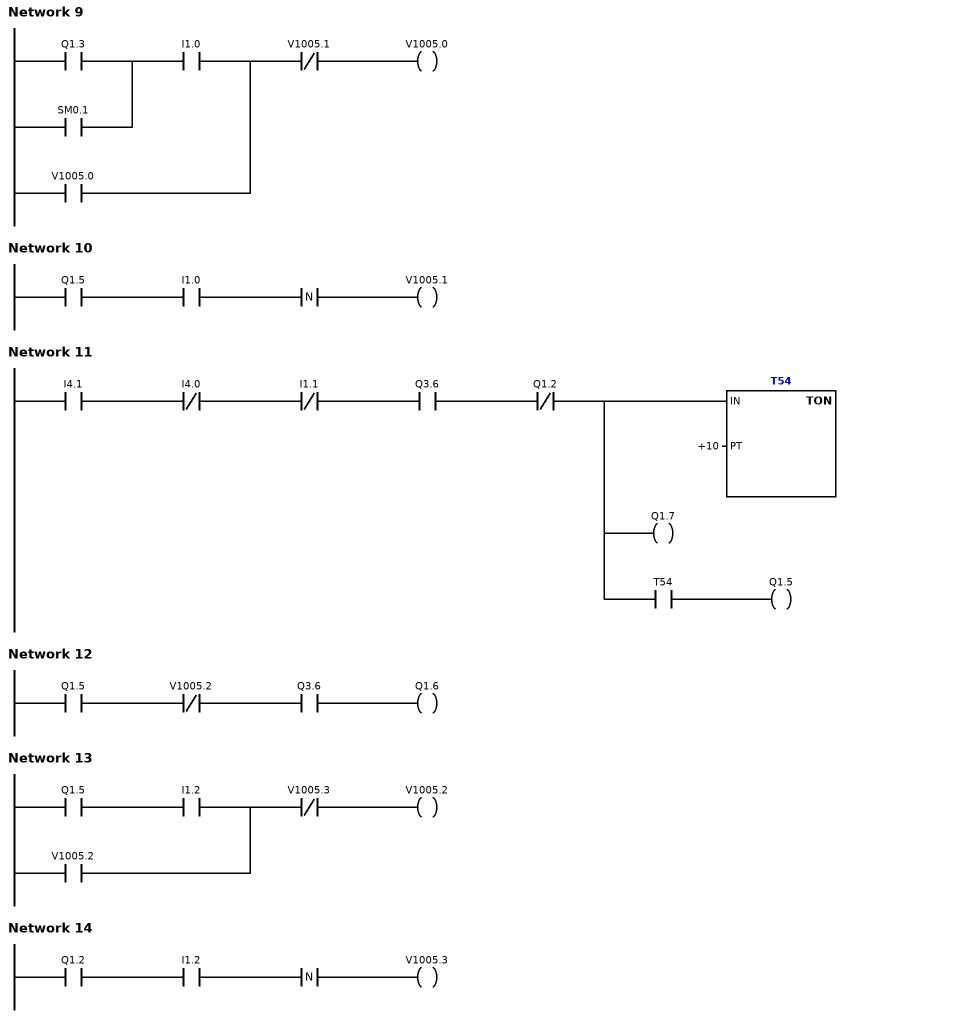
[picture p24: SBR7 networks 9-14]
Network 9
LD     Q1.3
O      SM0.1
A      I1.0
O      V1005.0
AN     V1005.1
=      V1005.0
Network 10
LD     Q1.5
A      I1.0
ED
=      V1005.1
Network 11
LD     I4.1
AN     I4.0
AN     I1.1
A      Q3.6
AN     Q1.2
TON    T54, +10
=      Q1.7
A      T54
=      Q1.5
Network 12
LD     Q1.5
AN     V1005.2
A      Q3.6
=      Q1.6
Network 13
LD     Q1.5
A      I1.2
O      V1005.2
AN     V1005.3
=      V1005.2
Network 14
LD     Q1.2
A      I1.2
ED
=      V1005.3
END_SUBROUTINE_BLOCK

SUBROUTINE_BLOCK Sheed_lead:SBR8
TITLE=
BEGIN
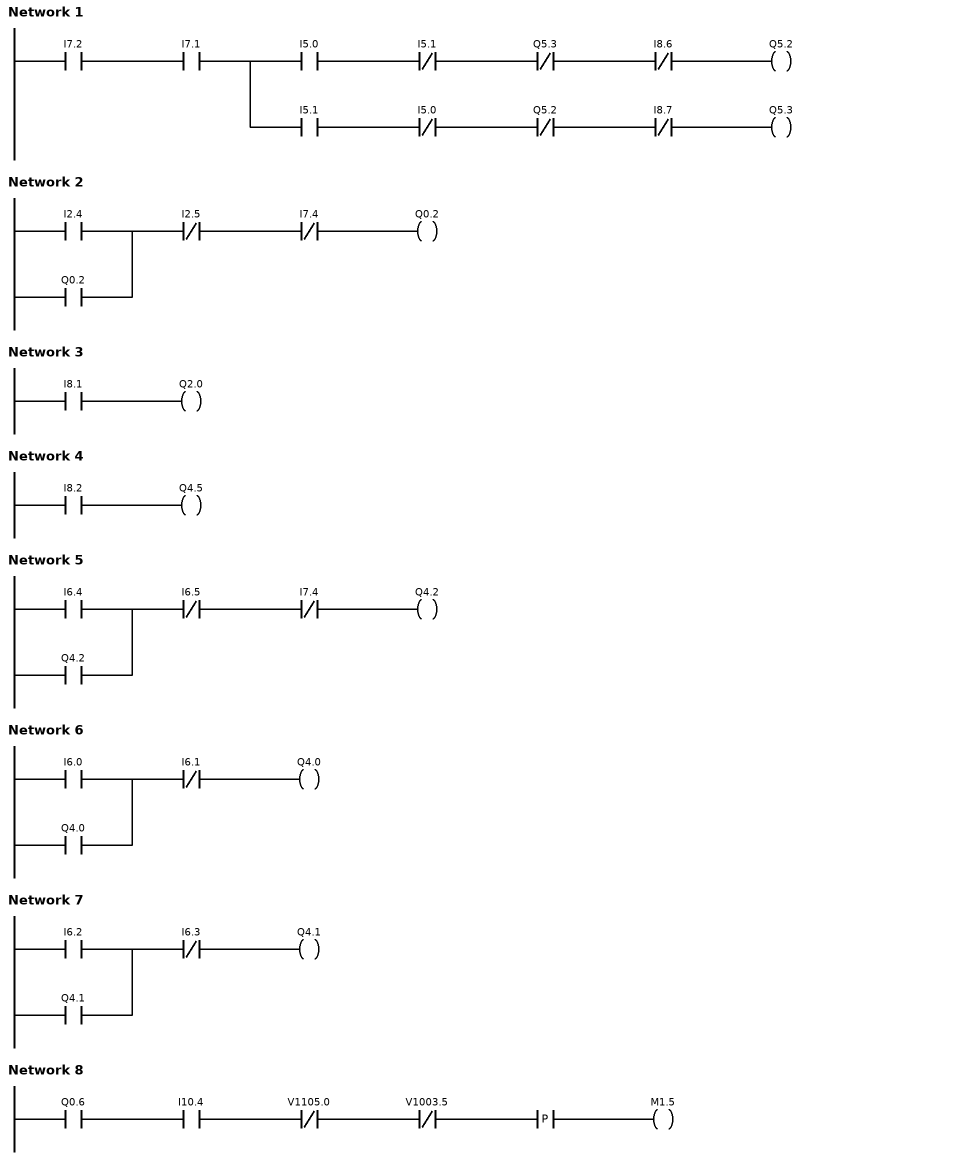
Network 1
LD     I7.2
A      I7.1
LPS
A      I5.0
AN     I5.1
AN     Q5.3
AN     I8.6
=      Q5.2
LPP
A      I5.1
AN     I5.0
AN     Q5.2
AN     I8.7
=      Q5.3
Network 2
LD     I2.4
O      Q0.2
AN     I2.5
AN     I7.4
=      Q0.2
Network 3
LD     I8.1
=      Q2.0
Network 4
LD     I8.2
=      Q4.5
Network 5
LD     I6.4
O      Q4.2
AN     I6.5
AN     I7.4
=      Q4.2
Network 6
LD     I6.0
O      Q4.0
AN     I6.1
=      Q4.0
Network 7
LD     I6.2
O      Q4.1
AN     I6.3
=      Q4.1
Network 8
LD     Q0.6
A      I10.4
AN     V1105.0
AN     V1003.5
EU
=      M1.5
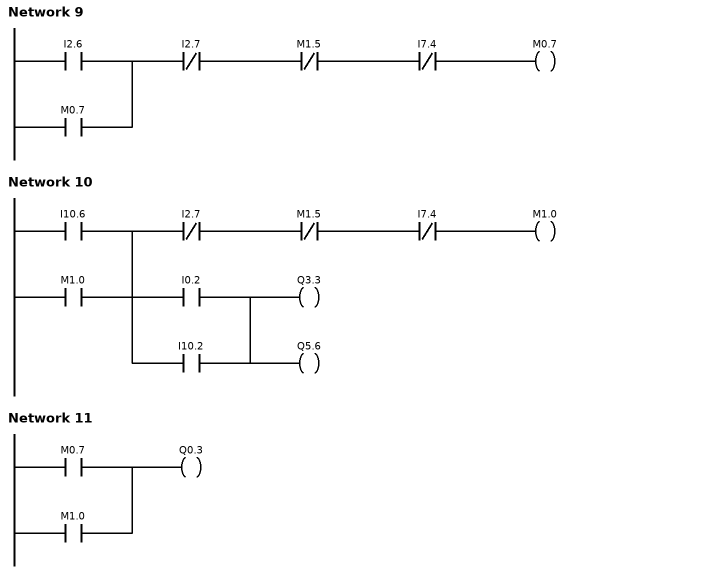
Network 9
LD     I2.6
O      M0.7
AN     I2.7
AN     M1.5
AN     I7.4
=      M0.7
Network 10
LD     I10.6
O      M1.0
LPS
AN     I2.7
AN     M1.5
AN     I7.4
=      M1.0
LPP
LD     I0.2
O      I10.2
ALD
=      Q3.3
=      Q5.6
Network 11
LD     M0.7
O      M1.0
=      Q0.3
END_SUBROUTINE_BLOCK

SUBROUTINE_BLOCK Core_Chuck:SBR9
TITLE=
BEGIN
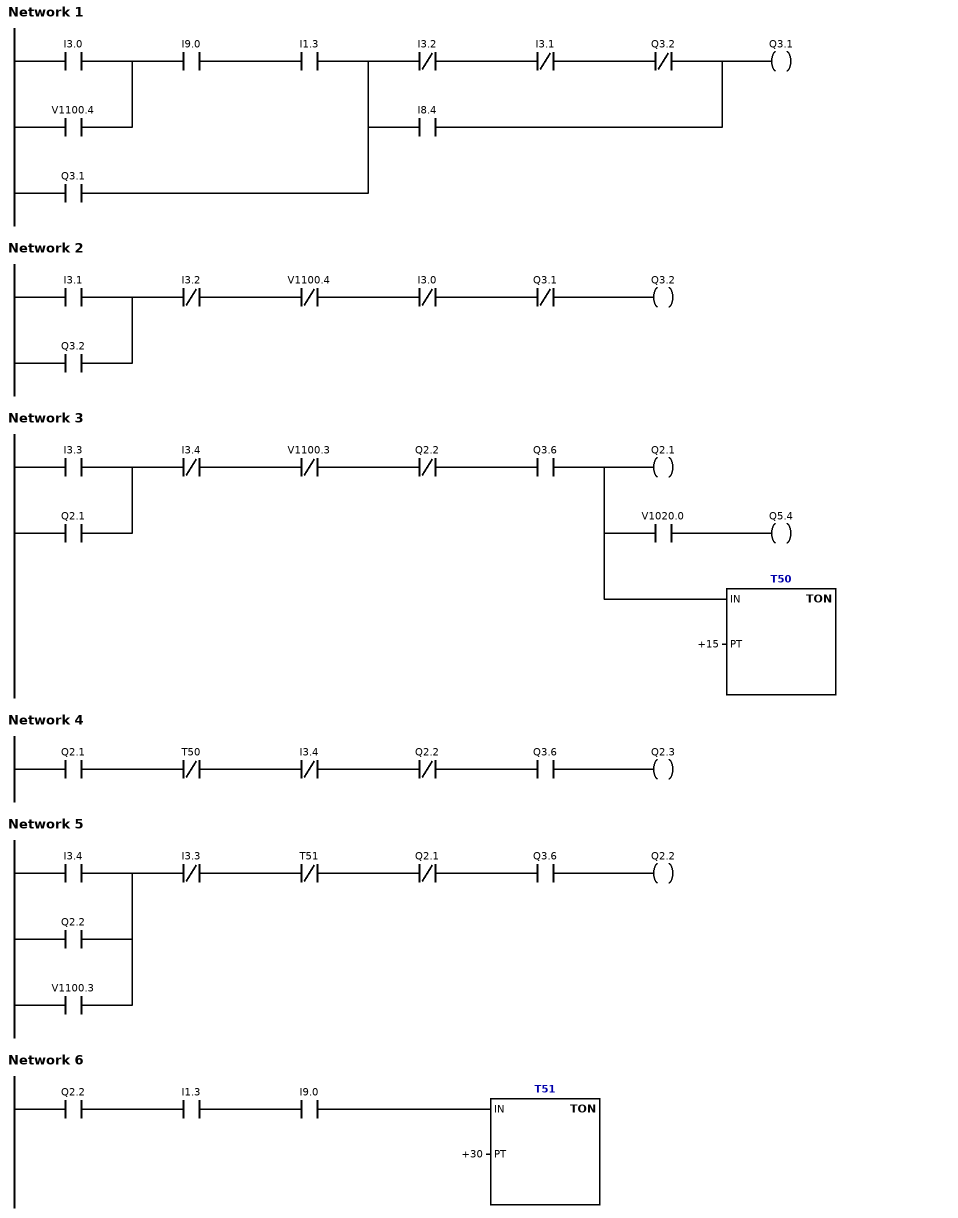
Network 1
LD     I3.0
O      V1100.4
A      I9.0
A      I1.3
O      Q3.1
LDN    I3.2
AN     I3.1
AN     Q3.2
O      I8.4
ALD
=      Q3.1
Network 2
LD     I3.1
O      Q3.2
AN     I3.2
AN     V1100.4
AN     I3.0
AN     Q3.1
=      Q3.2
Network 3
LD     I3.3
O      Q2.1
AN     I3.4
AN     V1100.3
AN     Q2.2
A      Q3.6
LPS
=      Q2.1
A      V1020.0
=      Q5.4
LPP
TON    T50, +15
Network 4
LD     Q2.1
AN     T50
AN     I3.4
AN     Q2.2
A      Q3.6
=      Q2.3
Network 5
LD     I3.4
O      Q2.2
O      V1100.3
AN     I3.3
AN     T51
AN     Q2.1
A      Q3.6
=      Q2.2
Network 6
LD     Q2.2
A      I1.3
A      I9.0
TON    T51, +30
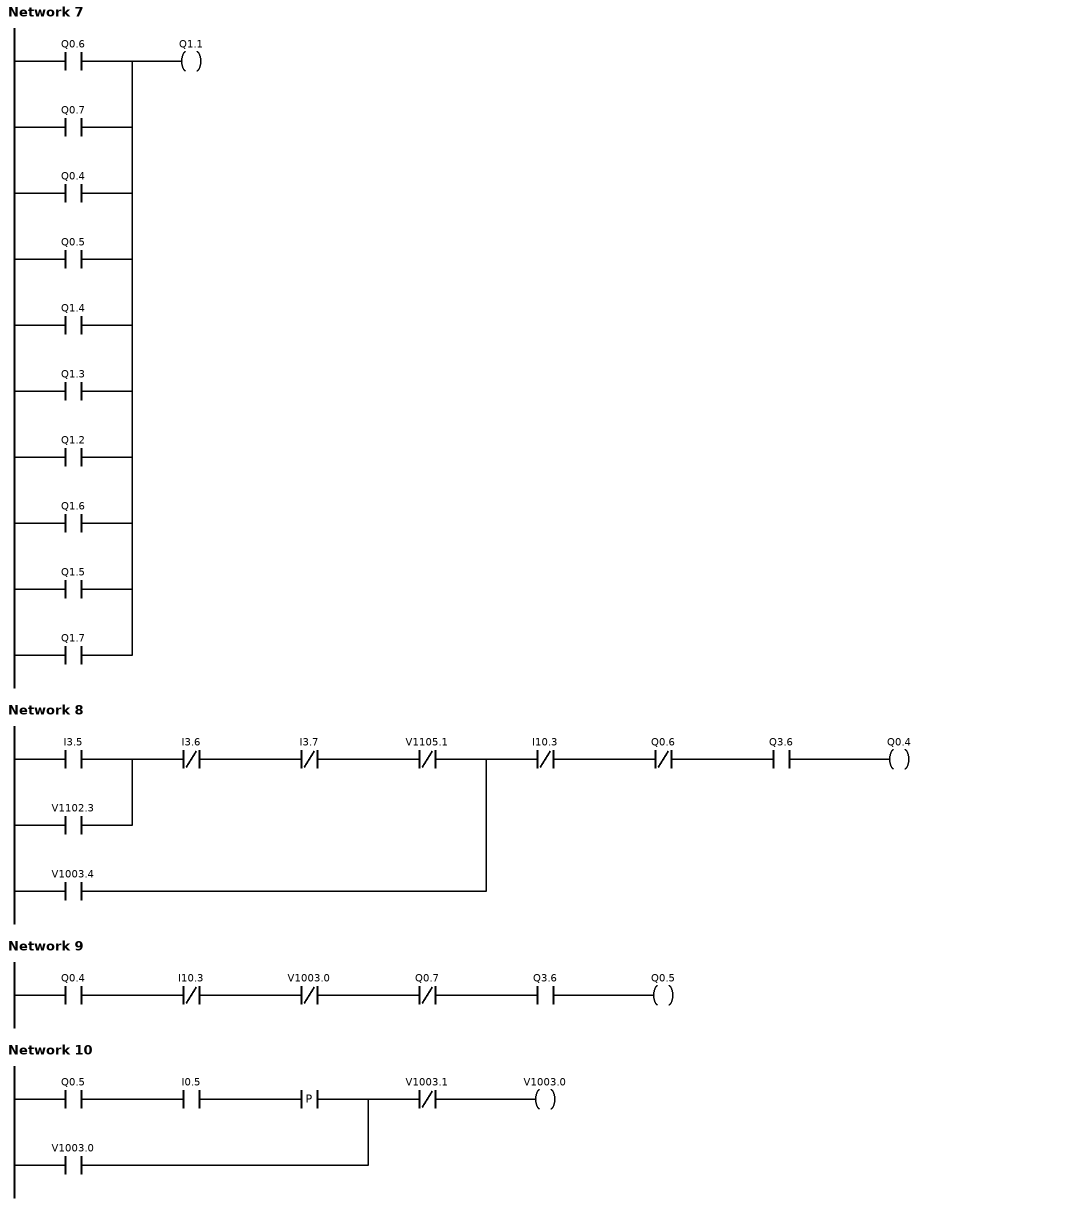
Network 7
LD     Q0.6
O      Q0.7
O      Q0.4
O      Q0.5
O      Q1.4
O      Q1.3
O      Q1.2
O      Q1.6
O      Q1.5
O      Q1.7
=      Q1.1
Network 8
LD     I3.5
O      V1102.3
AN     I3.6
AN     I3.7
AN     V1105.1
O      V1003.4
AN     I10.3
AN     Q0.6
A      Q3.6
=      Q0.4
Network 9
LD     Q0.4
AN     I10.3
AN     V1003.0
AN     Q0.7
A      Q3.6
=      Q0.5
Network 10
LD     Q0.5
A      I0.5
EU
O      V1003.0
AN     V1003.1
=      V1003.0
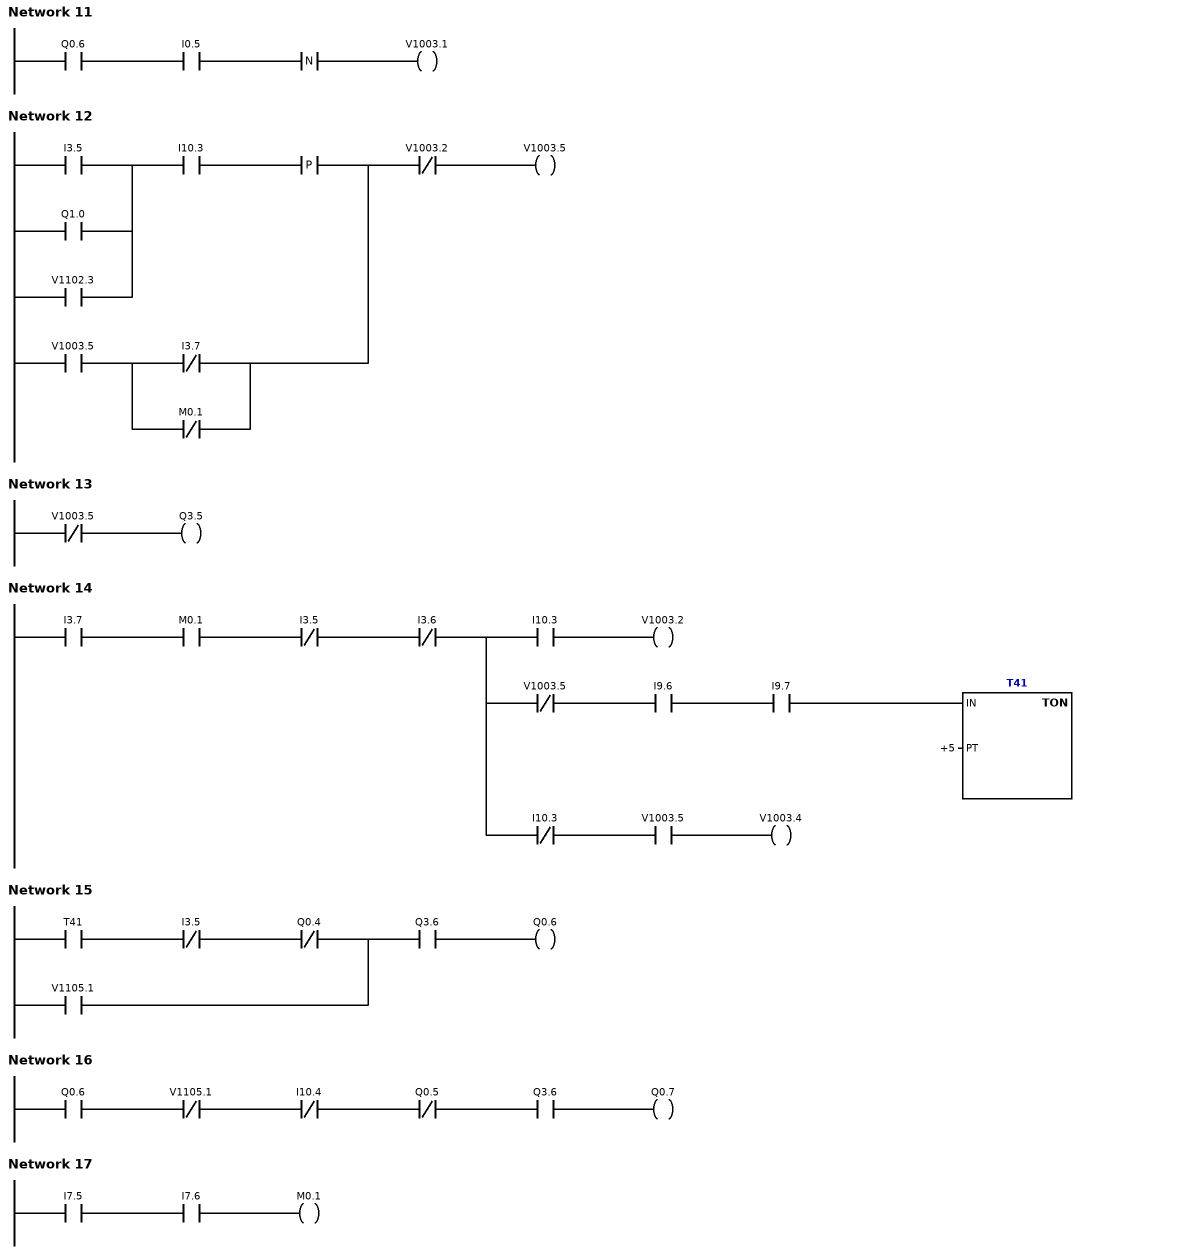
Network 11
LD     Q0.6
A      I0.5
ED
=      V1003.1
Network 12
LD     I3.5
O      Q1.0
O      V1102.3
A      I10.3
EU
LD     V1003.5
LDN    I3.7
ON     M0.1
ALD
OLD
AN     V1003.2
=      V1003.5
Network 13
LDN    V1003.5
=      Q3.5
Network 14
LD     I3.7
A      M0.1
AN     I3.5
AN     I3.6
LPS
A      I10.3
=      V1003.2
LRD
AN     V1003.5
A      I9.6
A      I9.7
TON    T41, +5
LPP
AN     I10.3
A      V1003.5
=      V1003.4
Network 15
LD     T41
AN     I3.5
AN     Q0.4
O      V1105.1
A      Q3.6
=      Q0.6
Network 16
LD     Q0.6
AN     V1105.1
AN     I10.4
AN     Q0.5
A      Q3.6
=      Q0.7
Network 17
LD     I7.5
A      I7.6
=      M0.1
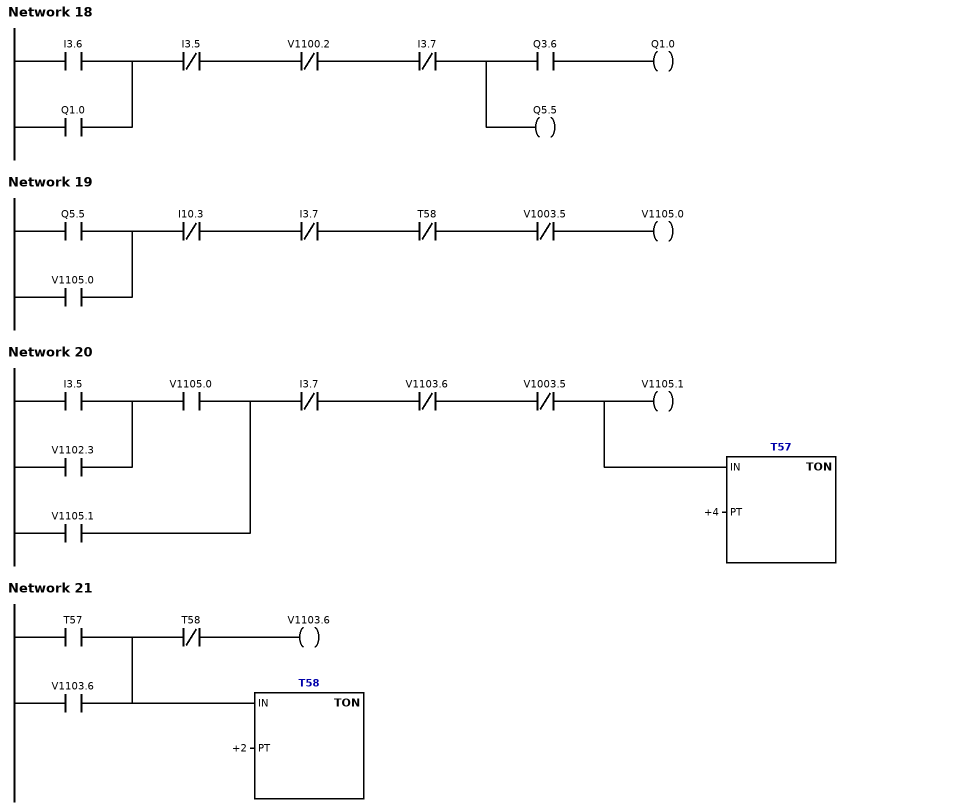
Network 18
LD     I3.6
O      Q1.0
AN     I3.5
AN     V1100.2
AN     I3.7
LPS
A      Q3.6
=      Q1.0
LPP
=      Q5.5
Network 19
LD     Q5.5
O      V1105.0
AN     I10.3
AN     I3.7
AN     T58
AN     V1003.5
=      V1105.0
Network 20
LD     I3.5
O      V1102.3
A      V1105.0
O      V1105.1
AN     I3.7
AN     V1103.6
AN     V1003.5
=      V1105.1
TON    T57, +4
Network 21
LD     T57
O      V1103.6
LPS
AN     T58
=      V1103.6
LPP
TON    T58, +2
END_SUBROUTINE_BLOCK

SUBROUTINE_BLOCK Value_1:SBR10
TITLE=
VAR_INPUT
d1:REAL;	// LD0 
H:REAL;	// LD4 
END_VAR
VAR_OUTPUT
D:REAL;	// LD8 
END_VAR
BEGIN
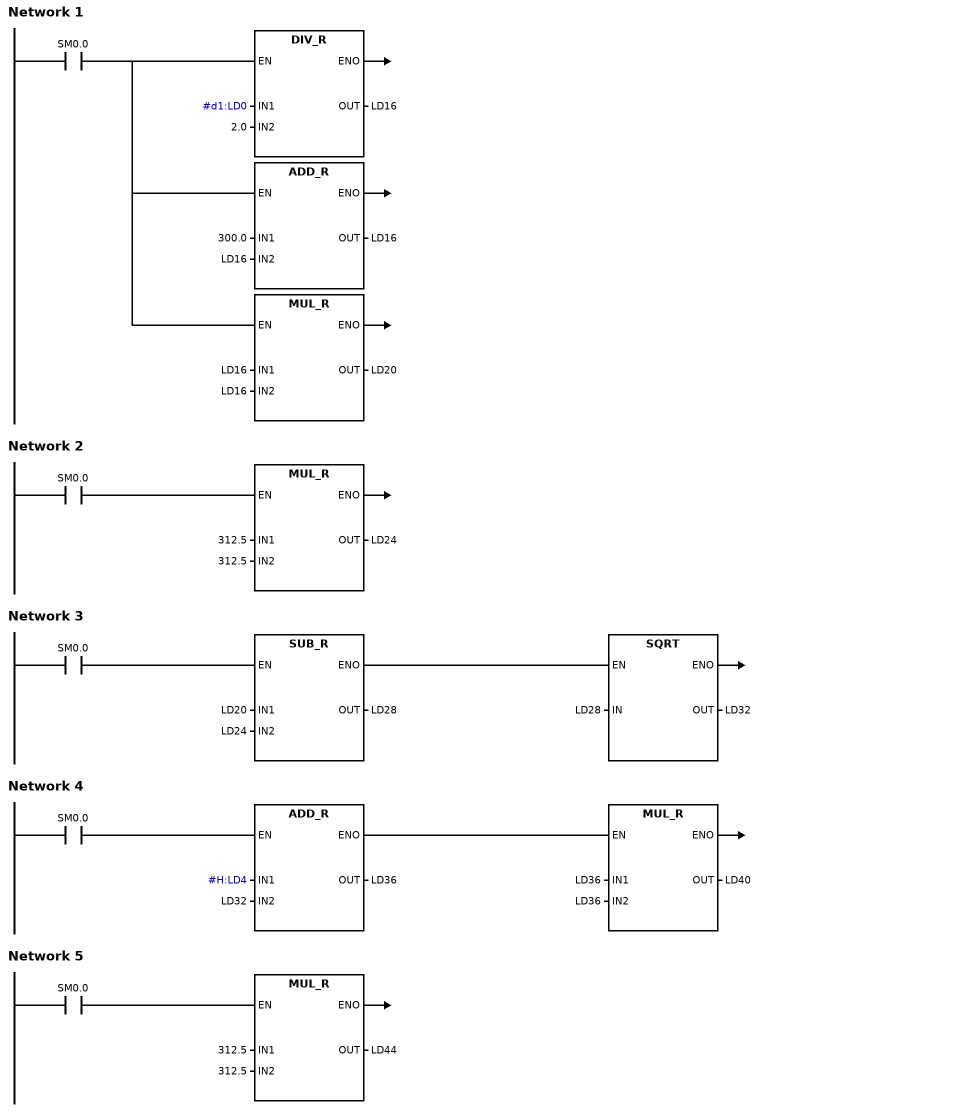
Network 1
LD     SM0.0
MOVR   #d1:LD0, LD16
/R     2.0, LD16
+R     300.0, LD16
MOVR   LD16, LD20
*R     LD16, LD20
Network 2
LD     SM0.0
MOVR   312.5, LD24
*R     312.5, LD24
Network 3
LD     SM0.0
MOVR   LD20, LD28
AENO
-R     LD24, LD28
AENO
SQRT   LD28, LD32
Network 4
LD     SM0.0
MOVR   #H:LD4, LD36
AENO
+R     LD32, LD36
AENO
MOVR   LD36, LD40
*R     LD36, LD40
Network 5
LD     SM0.0
MOVR   312.5, LD44
*R     312.5, LD44
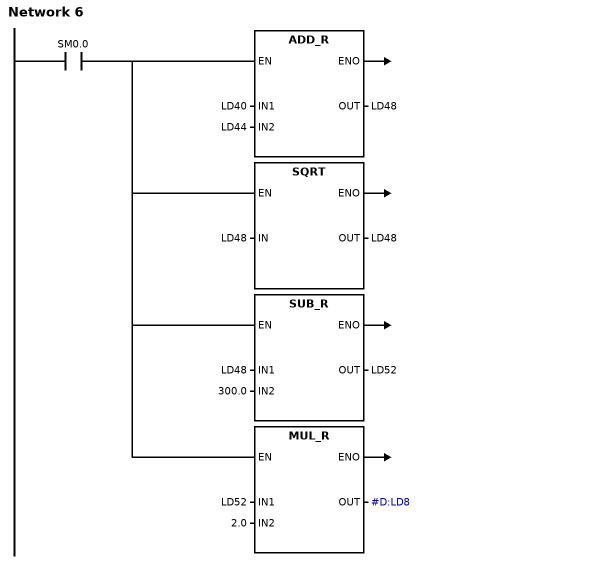
Network 6
LD     SM0.0
MOVR   LD40, LD48
+R     LD44, LD48
SQRT   LD48, LD48
MOVR   LD48, LD52
-R     300.0, LD52
MOVR   LD52, #D:LD8
*R     2.0, #D:LD8
END_SUBROUTINE_BLOCK

SUBROUTINE_BLOCK TOSHIBA_DO:SBR11
TITLE=
BEGIN
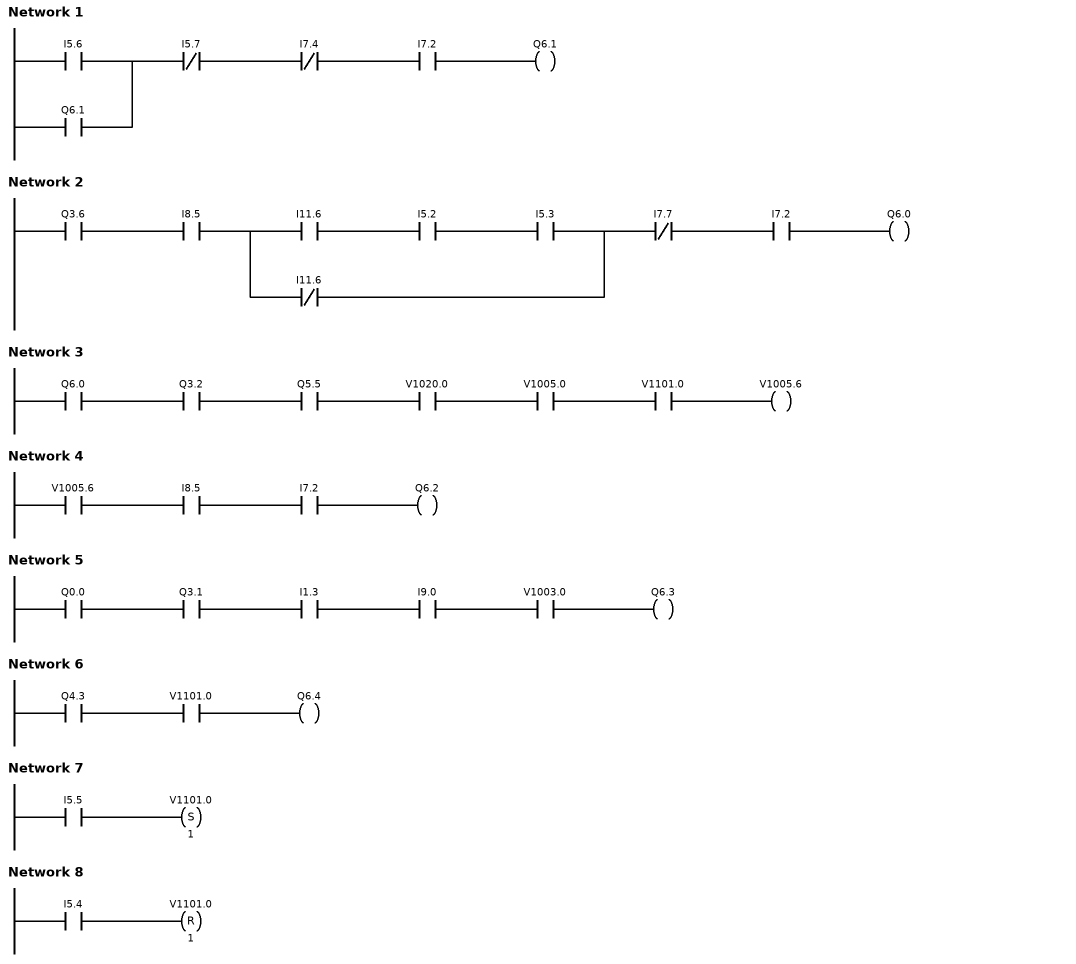
Network 1
LD     I5.6
O      Q6.1
AN     I5.7
AN     I7.4
A      I7.2
=      Q6.1
Network 2
LD     Q3.6
A      I8.5
LD     I11.6
A      I5.2
A      I5.3
ON     I11.6
ALD
AN     I7.7
A      I7.2
=      Q6.0
Network 3
LD     Q6.0
A      Q3.2
A      Q5.5
A      V1020.0
A      V1005.0
A      V1101.0
=      V1005.6
Network 4
LD     V1005.6
A      I8.5
A      I7.2
=      Q6.2
Network 5
LD     Q0.0
A      Q3.1
A      I1.3
A      I9.0
A      V1003.0
=      Q6.3
Network 6
LD     Q4.3
A      V1101.0
=      Q6.4
Network 7
LD     I5.5
S      V1101.0, 1
Network 8
LD     I5.4
R      V1101.0, 1
END_SUBROUTINE_BLOCK

SUBROUTINE_BLOCK Auto_Roll_Eiector:SBR12
TITLE=
BEGIN
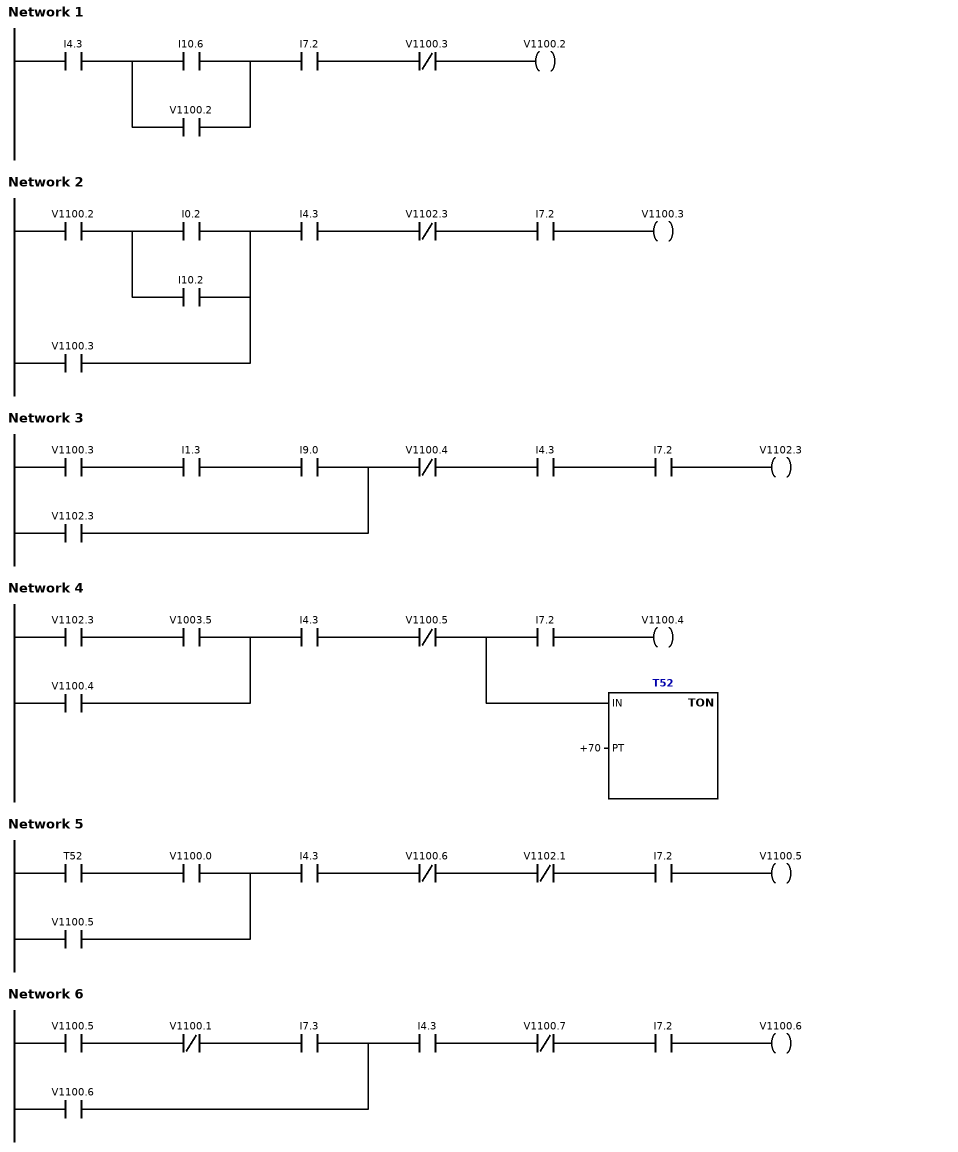
Network 1
LD     I4.3
LD     I10.6
O      V1100.2
ALD
A      I7.2
AN     V1100.3
=      V1100.2
Network 2
LD     V1100.2
LD     I0.2
O      I10.2
ALD
O      V1100.3
A      I4.3
AN     V1102.3
A      I7.2
=      V1100.3
Network 3
LD     V1100.3
A      I1.3
A      I9.0
O      V1102.3
AN     V1100.4
A      I4.3
A      I7.2
=      V1102.3
Network 4
LD     V1102.3
A      V1003.5
O      V1100.4
A      I4.3
AN     V1100.5
LPS
A      I7.2
=      V1100.4
LPP
TON    T52, +70
Network 5
LD     T52
A      V1100.0
O      V1100.5
A      I4.3
AN     V1100.6
AN     V1102.1
A      I7.2
=      V1100.5
Network 6
LD     V1100.5
AN     V1100.1
A      I7.3
O      V1100.6
A      I4.3
AN     V1100.7
A      I7.2
=      V1100.6
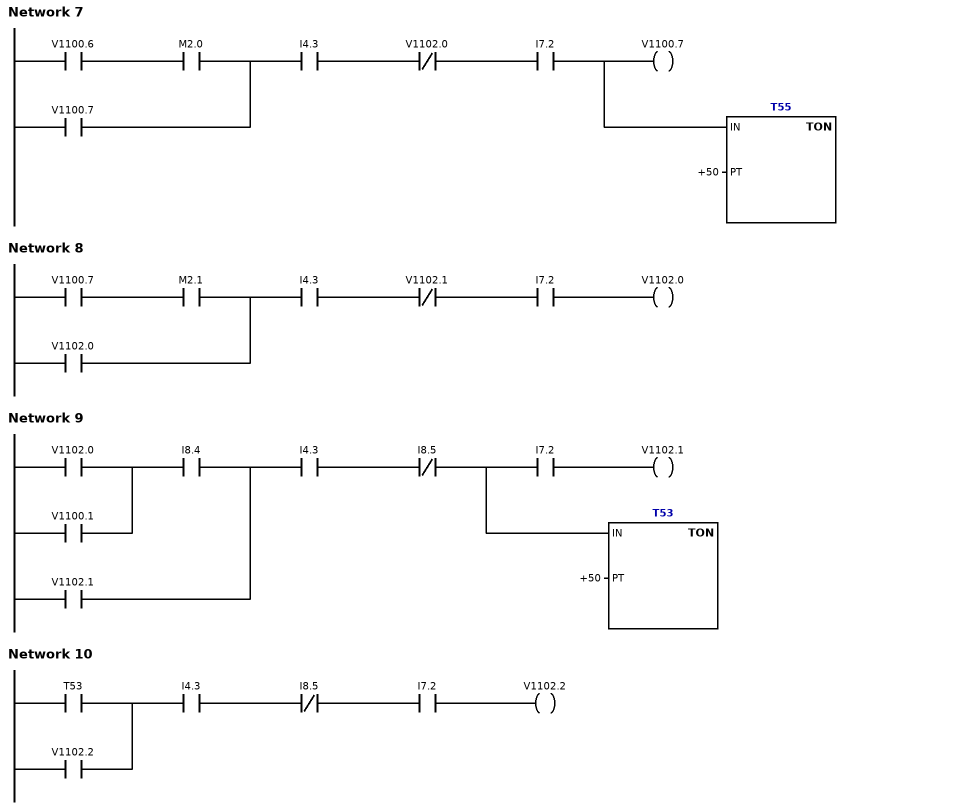
Network 7
LD     V1100.6
A      M2.0
O      V1100.7
A      I4.3
AN     V1102.0
A      I7.2
=      V1100.7
TON    T55, +50
Network 8
LD     V1100.7
A      M2.1
O      V1102.0
A      I4.3
AN     V1102.1
A      I7.2
=      V1102.0
Network 9
LD     V1102.0
O      V1100.1
A      I8.4
O      V1102.1
A      I4.3
AN     I8.5
LPS
A      I7.2
=      V1102.1
LPP
TON    T53, +50
Network 10
LD     T53
O      V1102.2
A      I4.3
AN     I8.5
A      I7.2
=      V1102.2
END_SUBROUTINE_BLOCK

SUBROUTINE_BLOCK TOSHIBA_Diameter_AO:SBR13
TITLE=
VAR_INPUT
temp0:REAL;	// LD0 
END_VAR
VAR_OUTPUT
temp6:REAL;	// LD4 
END_VAR
BEGIN
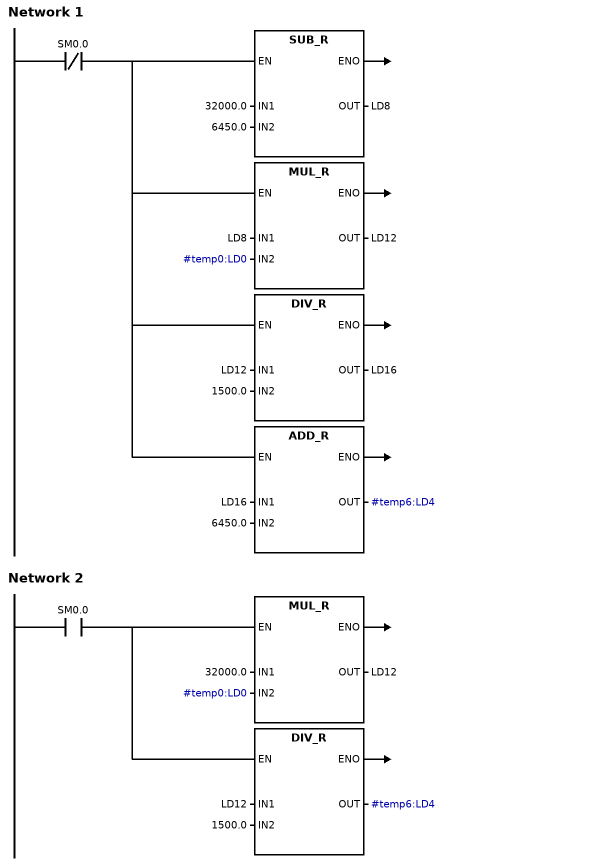
Network 1
LDN    SM0.0
MOVR   32000.0, LD8
-R     6450.0, LD8
MOVR   LD8, LD12
*R     #temp0:LD0, LD12
MOVR   LD12, LD16
/R     1500.0, LD16
MOVR   LD16, #temp6:LD4
+R     6450.0, #temp6:LD4
Network 2
LD     SM0.0
MOVR   32000.0, LD12
*R     #temp0:LD0, LD12
MOVR   LD12, #temp6:LD4
/R     1500.0, #temp6:LD4
END_SUBROUTINE_BLOCK

SUBROUTINE_BLOCK System_fault:SBR14
TITLE=
BEGIN
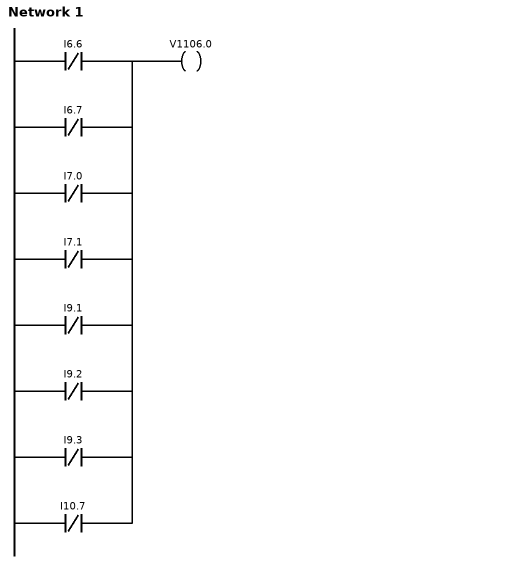
Network 1
LDN    I6.6
ON     I6.7
ON     I7.0
ON     I7.1
ON     I9.1
ON     I9.2
ON     I9.3
ON     I10.7
=      V1106.0
END_SUBROUTINE_BLOCK
